/// container for all communication data types that are used by the unit
TYPE HandlingComRef :
STRUCT
  Publish : REFERENCE TO HandlingComPublish; 
  Subscribe : REFERENCE TO HandlingComSubscribe; 
END_STRUCT
END_TYPE

(* stored: Version 1.1.0.1
   DUT HandlingComRef: Id {97f0b3f6-7f91-4ac1-9dac-181a313ed230} *)
